// TIA Portal V18 export
TYPE "MEStoPLC_ProcessingExchange"
// stored: IsFailsafeCompliant false
   STRUCT
      "M-ProcessingDone" : Bool;   // 记录ID，标记不能重复加工，
      Reserve : Array[1..298] of Byte;   // Processing交互预留
   END_STRUCT;
END_TYPE
